TYPE EnableXonXoffTx EXTENDS SubIndexModuleBase :
STRUCT
END_STRUCT
END_TYPE

(* stored: Version 1.1.0.1, ProductVersion 3.1.4024.3
   DUT EnableXonXoffTx: Id {ad4eabff-6fa6-462d-b645-7775b2f0c4dc} *)
